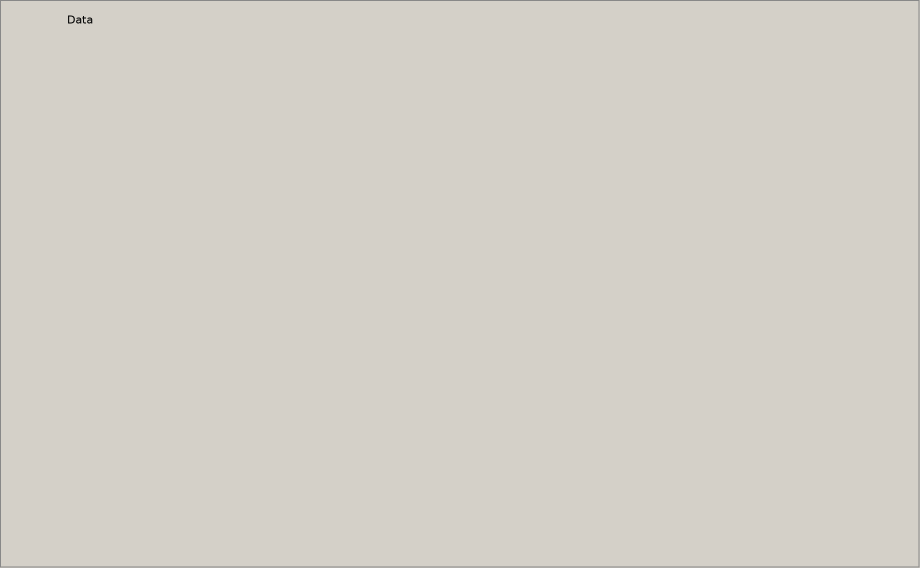
VISUALIZATION Data  // 920x568
    Label (5,5 150x30), "Data"
END_VISUALIZATION

(* stored: Version 1.1.0.1
   Visu Data: Id {1bbe9ea3-3968-45ad-b6a7-b6754c0a0375} *)
